{attribute 'reflection'}
FUNCTION_BLOCK FB_PitchControlOld
VAR_IN_OUT
	Pitch : HOMS_PitchMechanismOld;
END_VAR
VAR_INPUT
	DirectPiezoMode	:	BOOL := FALSE; //Set this true to tell the piezo what position to seek in closed loop
	rReqAbsPos	:	REAL; //Control the pitch position with this when DirectPiezoMode is false
END_VAR
VAR_OUTPUT
	q_xError	:	BOOL;
	q_xDone	:	BOOL;
	q_xBusy	:	BOOL;
END_VAR
VAR
	//Introspection
	//////////////////////////////
		{attribute 'instance-path'}
		{attribute 'no_init'}
		POUName	:	STRING; //Name of the POU for logging/error reporting
	
	
	//FB Boilerplate
	//////////////////////
		stDiag	:	ST_fbDiagnostics;
		fbFormatString	:	FB_FormatString;
		
	//Working variables
	/////////////////////////
		PC_State 		:	E_PitchControl := PCM_Init;
		rPrevReqAbsPos	:	REAL; //Previously  requested abs position
		rPrevStepperPos :	REAL; //Previously successfully achieved stepper position
		tonStepperHold	:	TON := (PT := T#100MS); //Timer to hold stepper position while the system relaxes
		FirstPass	:	BOOL := TRUE; //set false after first pass, used for initializations
		Coarse50PiezoMove	:	BOOL;
		OriginalPosRequest: REAL;
		//PTP
		/////////////////////////
				Drive         : FB_DRIVE;
				fbCoE         : FB_ElmoGDCBellCoE;
				nCommand      : UINT;
				rLastSetpoint : REAL;
				rtTweakFwd    : R_TRIG;
				rtTweakBwd    : R_TRIG;
				rtExecute     : R_TRIG;
				bRequesting   : BOOL;
				rSetpoint     : REAL; //Adjusted based on abs pos request or tweaks.
				mcSmoothMover	:	MC_SmoothMover;
	
	//Axis Control Blocks
	/////////////////////////////
		fbPiezoControl	:	FB_PiezoControl;
	
	
	//Triggers
	//////////////////////////////
		rtManualMode:	R_TRIG;
		ftManualMode	:	F_TRIG;
		rtStepperDone	:	R_TRIG;

	lrActPos: LREAL;
	tonPiezoSettled	: TON := (PT:=T#2S);
	tonPiezoDone	:	TON := (PT:=T#500ms);
	
	ftLimitSwitch: F_TRIG;
	// Flag to track when a limit switch has been hit.
	xLimitHit: BOOL;
	rtPiezoMoveDone: R_TRIG;
	rtHalt: R_TRIG;
	bCoarseMoveComplete	:	BOOL; //Set after a coarse move completes, added because coarse moves can be interrupted
END_VAR
VAR CONSTANT
	cPiezoRange	:	REAL := 60; // 90um of stroke to the piezo, which means a 180urad stroke...
    cOperatingRegion : REAL := 0.75; // Only use a fraction of the piezo range before forcing a coarse move    
END_VAR

(* HOMS Pitch Control
A. Wallace

The HOMS Pitch mechanism consists of a stepper and piezo that work together to adjust
the pitch of the mirror assembly.

Pitch control state machine

If the target position is beyond the range of the piezo mechanism,
execute a coarse pitch move with the stepper. 
The target of the coarse move shall be set to the requested position. 
Once coarse motion has completed the coarse motion drive position 
correction output shall be set to zero.

Fine pitch motion with the piezo will be initiated to finish closing the loop.

The piezo mechanism can actuate ~ 180urad or 90um.

*)

lrActPos := Pitch.Stepper.stAxis.NcToPlc.ActPos;
nCommand  := 3;
(* If we hit a limit during a move, we need to change the setpoint *)
ftLimitSwitch(CLK:=Pitch.Stepper.xHiLS AND Pitch.Stepper.xLoLS);

//Manual mode switching logic
/////////////////////////////////////
	rtManualMode(CLK:=DirectPiezoMode);
	ftManualMode(CLK:=DirectPiezoMode);
	A_ModeSwitch();

//Motion control logic from PTP	
//Tweak Triggers
/////////////////////////////////////////////
	rtTweakFwd(CLK:=Pitch.Axis.bTwkFwd);
	rtTweakBwd(CLK:=Pitch.Axis.bTwkBwd);
	rtExecute(CLK:=NOT Pitch.Stepper.stAxis.Status.NotMoving);
	
//Tweak Forward
/////////////////////
IF rtTweakFwd.Q THEN
	//Setup move
	Pitch.Axis.rReqAbsPos := rLastSetpoint + Pitch.Axis.rTweak;
//Tweak Backwards
/////////////////////
ELSIF rtTweakBwd.Q THEN
	//Setup move
	Pitch.Axis.rReqAbsPos := rLastSetpoint - Pitch.Axis.rTweak;
ELSE
	bRequesting := FALSE;
END_IF

(* At this point, Pitch.Axis.rReqAbsPos holds the next setpoint.
Now it will be validated against the soft-limits
*)

//Halt
///////////////////////////////////
	rtHalt(CLK:= Pitch.Axis.xStop);
	(* Halt does the following
	Halts stepper motion, waits for stepper to settle, records stepper position as prev. stepper pos.
	moves to fine move with a new abs setpoint
	*)
	IF rtHalt.Q AND NOT q_xDone THEN
		PC_State := PCM_Halt;
	END_IF

//Check for new position requests, and sanitize
///////////////////////////////////////////////
	IF (rLastSetpoint <> Pitch.Axis.rReqAbsPos) THEN
		//We don't want to initiate any kind of a move if we don't have to.
		IF 	Pitch.Axis.rReqAbsPos > Pitch.ReqPosLimHi OR Pitch.Axis.rReqAbsPos < Pitch.ReqPosLimLo OR
			(Pitch.Axis.rReqAbsPos < lrActPos) AND Pitch.Axis.xLoLS OR (Pitch.Axis.rReqAbsPos > lrActPos) AND Pitch.Axis.xHiLS THEN
			//Requested move is outside of travel limits
			OriginalPosRequest	:= Pitch.Axis.rReqAbsPos;
			Pitch.Axis.rReqAbsPos := LIMIT(Pitch.ReqPosLimLo, Pitch.Axis.rReqAbsPos, Pitch.ReqPosLimHi);
			//Only want to log one warning about a bad position request.
			IF OriginalPosRequest <> Pitch.Axis.rReqAbsPos THEN
				//Log a warning
				fbFormatString.sFormat := 'Pitch req OoR fb (%s), reset within limits, %f';
				fbFormatString.arg1 := F_STRING(POUName);
				fbFormatString.arg2 := F_REAL(OriginalPosRequest);
				//fbFormatString(sOut=>fbLogMessage.i_sMsg);
				fbFormatString(sOut=>stDiag.asResults[stDiag.resultIdx.IncVal()]);
				//fbLogMessage(i_eSevr:= Warning, i_eSubsystem:=gDefaultSubsystem);
			END_IF
		END_IF
		// At this point Pitch.Axis.rReqAbsPos is considered clean and safe, so we pass to a holding variable
		rSetpoint := Pitch.Axis.rReqAbsPos;
		//Set the previously requested position here
		rLastSetpoint := rSetpoint;
		//New position request, no longer done.
		q_xDone := FALSE;
		q_xBusy	:= TRUE;
		PC_State := PCM_MoveRequested;
	END_IF
	
//State Machine
//////////////////////////////////
CASE PC_State OF
	PCM_Init: 
		//Initialize stepper motor mc power block
		Drive.bReset := FirstPass;
		PC_State := PCM_Standby;
		
	PCM_Standby:
		;
		
	PCM_MoveRequested: 
		//A move has been requested, is it within range of the piezo?
		IF WithinRange(ValA:=rSetpoint, Center:=rPrevStepperPos, Range:=cPiezoRange, Offset:=0)
                //Ensure that the piezo is not currently outside the operating range
                //Otherwise, force a coarse move that will rezero the piezo travel
	        AND WithinRange(ValA:=Pitch.Piezo.rActVoltage,
                                Center:=(Pitch.Piezo.LowerVoltage + Pitch.Piezo.UpperVoltage)/2.0,
                                Range:=cOperatingRegion*(Pitch.Piezo.UpperVoltage - Pitch.Piezo.LowerVoltage)/2.0,
                                Offset:=0)
			AND bCoarseMoveComplete
		THEN
			//Move is within the nominal range of the piezo
			fbFormatString.sFormat := 'Within range, fine move %f';
			fbFormatString.arg1 := F_REAL(rSetpoint);
			fbFormatString(sOut=>stDiag.asResults[stDiag.resultIdx.IncVal()]);
			PC_State := PCM_FineMove;
		ELSE
			// Out of range, head to coarse move
			fbFormatString.sFormat := 'OoR, using stepper %f';
			fbFormatString.arg1 := F_REAL(rSetpoint);
			fbFormatString(sOut=>stDiag.asResults[stDiag.resultIdx.IncVal()]);
			bCoarseMoveComplete := FALSE;
			PC_State := PCM_Coarse50Piezo;
		END_IF
		
	PCM_Coarse50Piezo:
		//A coarse move uses the stepper to do a best-effort position
		//First set the piezo to nominal 50% extension using idle mode
		//////////////////////////////////////////////////////////////////////////////
		Pitch.Piezo.xIdleMode := TRUE;
		//Indicate we are doing the coarse 50% piezo move	
		Coarse50PiezoMove := TRUE;
		//Wait for piezo to settle
		tonPiezoSettled.IN := TRUE;
		Coarse50PiezoMove R= tonPiezoSettled.Q;
		IF tonPiezoSettled.Q THEN
			//Piezo has moved to 50% position, finish with the stepper
			PC_State := PCM_CoarseMove;
			Pitch.Stepper.xEnable := TRUE;
			tonPiezoSettled.IN := FALSE;
		END_IF
		
	PCM_CoarseMove: 
		//With the piezo at a nom 50% extension, move the stepper to requested position
		IF Drive.bEnabled THEN
			//Drive.fPosition := rSetpoint;
			//Drive.bExecute := TRUE;
			
			mcSmoothMover.ReqAbsPos := rSetpoint;
			mcSmoothMover.Enable := TRUE;
		END_IF

		IF ftLimitSwitch.Q THEN
			Drive.fPosition := lrActPos;
			
			mcSmoothMover.ReqAbsPos := lrActPos;
			
			xLimitHit	:= TRUE; //set this flag here.
		END_IF
		tonStepperHold.IN := WithinRange(ValA:=LREAL_TO_REAL(lrActPos), Center:=rSetpoint, Range:=Pitch.Stepper.rStepperDmovRange, Offset:=0);
		tonStepperHold(); //call this here to reset Q just below on first cycle
		//If the coarse move is complete, finish position correction with the piezo
		IF tonStepperHold.Q  OR ftLimitSwitch.Q THEN
			PC_State := PCM_CoarseMoveCleanup;
		ELSIF Pitch.Stepper.stStatus.bError OR Drive.bError OR mcSmoothMover.Error THEN
			Drive.bExecute := FALSE;
			mcSmoothMover.Enable := FALSE;
			Pitch.Stepper.xEnable := FALSE;
			PC_State := PCM_StepperError;
			//Stepper fb has encountered an error, pass a message to the logger
			IF Pitch.Stepper.stStatus.bError THEN
				fbFormatString.sFormat := 'Coarse move error, stepper err id %d';
				fbFormatString.arg1 := F_UDINT(Pitch.Stepper.stStatus.nErrorId);
			ELSIF Drive.bError THEN
				fbFormatString.sFormat := 'Coarse move error, drive err id %d';
				fbFormatString.arg1 := F_UDINT(Drive.nErrorId);
			ELSIF mcSmoothMover.Error THEN
				fbFormatString.sFormat := 'Coarse move error, smoothmover error';
			END_IF
			fbFormatString(sOut=>stDiag.asResults[stDiag.resultIdx.IncVal()]);
		END_IF
		
	PCM_CoarseMoveCleanup:
		Drive.bExecute := FALSE;
		//Calling Drive with execute false will halt the axis
		//Once halted, the axis will be in standstill
		// then we can disble it without error.
		IF Pitch.Stepper.stAxis.Status.StandStill THEN
			Pitch.Stepper.xEnable := FALSE;
		END_IF
		IF Pitch.Stepper.stAxis.Status.Disabled THEN
			rPrevStepperPos := mcSmoothMover.ReqAbsPos;
			bCoarseMoveComplete	:= TRUE;
			PC_State := PCM_FineMove;
		END_IF

	PCM_FineMove:	
		Pitch.Piezo.xIdleMode := FALSE;
		fbPiezoControl.xExecute := TRUE;
		IF xLimitHit THEN
			Pitch.Piezo.rReqAbsPos := lrActPos;
		ELSE
			Pitch.Piezo.rReqAbsPos := rSetpoint;
		END_IF
		rtPiezoMoveDone(CLK:=fbPiezoControl.xDone);
		IF rtPiezoMoveDone.Q THEN
			fbPiezoControl.xExecute := FALSE;
			PC_State := PCM_Done;
		END_IF
		
	PCM_Halt:
		//We may transition to this state from anywhere, so we need to clean up and move to done
		//Halt the stepper
		//If trans. from FineMove, stepper is already disabled
		Drive.bExecute := FALSE;
		IF Pitch.Stepper.stAxis.Status.Standstill OR Pitch.Stepper.stAxis.Status.Disabled THEN
			Pitch.Stepper.xEnable := FALSE;
			//If the piezo control is done, we haven't started the fine move yet, so we can
			// record the current position as the prev. achv. stepper position.
			IF fbPiezoControl.xDone THEN
				rPrevStepperPos := lrActPos;
			END_IF
			// Very special case, where the setpoint is now where we halted
			rSetpoint := lrActPos;
			PC_State := PCM_FineMove;
		END_IF
		
	PCM_Done:
		
		Pitch.Axis.rReqAbsPos := rLastSetpoint; //this might be kind of funky
		xLimitHit := FALSE;
		//Indicate we're done
		q_xDone	:= TRUE;
		q_xBusy := FALSE;
		//Move back to standby
		PC_State := PCM_Standby;
	PCM_StepperError:
		Drive.bReset := TRUE; // set false again in PCM_Init
		q_xBusy := FALSE;
		PC_State := PCM_Init; 
	PCM_PiezoError:
		q_xBusy := FALSE;
		PC_State := PCM_Init;
	PCM_OtherError:
		q_xBusy := FALSE;
		PC_State := PCM_Init;
	
END_CASE

FirstPass := FALSE;

//Transfer the other stuff to the piezo
/////////////////////////////////////////
Pitch.Piezo.rActPos := lrActPos;

//Function blocks
ACT_PTP();

tonPiezoSettled();
tonStepperHold();

fbPiezoControl(iq_Piezo:=Pitch.Piezo,
	Enable_Positive:=Pitch.Stepper.xHiLS,
	Enable_Negative:=Pitch.Stepper.xLoLS
);

ACTION A_ModeSwitch:
(* When switching between modes, we need to make sure all the executes/ mode switches, etc. are cleared *)

// Automatic to manual
/////////////////////////////
IF rtManualMode.Q THEN
;
END_IF

// Manual to automatic
//////////////////////////////
IF ftManualMode.Q THEN
	;
END_IF
END_ACTION

ACTION ACT_PTP:
//Read CoE Parameters
/////////////////////////
fbCoE(stCoE:=Pitch.Stepper.stCoE);

//Give control of the axis to the Drive function block
///////////////////////////////////////////////////////
Drive(bEnable  := Pitch.Stepper.xEnable,
	  Axis     := Pitch.Stepper.stAxis,
	  nCommand := nCommand,
	  fAcceleration := Pitch.Stepper.fAcceleration,
	  fDeceleration := Pitch.Stepper.fDeceleration,
	  fVelocity     := Pitch.Stepper.fVelocity,
	  bLimitFwd     := Pitch.Stepper.xHiLS,
	  bLimitBwd     := Pitch.Stepper.xLoLS,
	  bDone	=>  Pitch.Stepper.bDone,
	  bBusy => Pitch.Stepper.bBusy,
	  stStepperStatus => Pitch.Stepper.stStatus
	  );

//Reset Execute to wait for next motion command
////////////////////////////////////////////////
//bExecute R= Drive.Status.NotMoving AND NOT bRequesting;

//MC Smooth Mover
////////////////////////////////////////////////
(* You can control an axis with MC blocks other than those in PTP or drive.
We just use the drive/PTP block to initialize the axis and manage the limit
switch logic *)
mcSmoothMover(Axis:=Pitch.Stepper.stAxis,
	Velocity:=Pitch.Stepper.fVelocity);
END_ACTION

END_FUNCTION_BLOCK

(* stored: Version 1.1.0.1, ProductVersion 3.1.4022.18
   POU FB_PitchControlOld: Id {157a40f4-fb3c-4f04-8b9b-6aa8032367b0}, SpecialFunc None
   Action A_ModeSwitch: Id {281d1c4f-e2d3-47e0-b22b-e39b29c10c9c}
   Action ACT_PTP: Id {567d6566-63fe-4281-a3e1-a243f492c380} *)
